FUNCTION TryConvert_BOOL_TO_TOD : BOOL
VAR_INPUT
	in : BOOL;
	out : REFERENCE TO TOD;
END_VAR

out := BOOL_TO_TOD(in);
TryConvert_BOOL_TO_TOD := TRUE;

END_FUNCTION

(* stored: Version 1.1.0.1, ProductVersion 3.1.4024.12
   POU TryConvert_BOOL_TO_TOD: Id {5201db1a-ae2d-4d07-894e-05b7126044a1}, SpecialFunc None *)
